PROGRAM P_MotorControl
VAR
	
  	error:BOOL;
    fJogVelocity :LREAL;
	MC_Halt_ServoB: MC_Halt;
	MC_Halt_ServoA: MC_Halt;
	sinGen : FB_singen;	
	ServoA_SPGen: FB_useExtSetpointGen;
	ServoB_SPGen: FB_useExtSetpointGen;
	nSawSPError : INT :=0;
	r_trig_0: r_trig;


	
	b_ExecuteGearIn: BOOL;
	MC_GearInA: MC_GearIn;
	MC_MoveRelativeA: MC_MoveRelative;
	bAbsMoveBExecute: BOOL;
	MC_MoveAbsolute_A: MC_MoveContinuousAbsolute;
	ZeroingReqRtrig: R_TRIG;
	bSetZero: BOOL;
	McWritePArams1: MC_WriteParameterPersistent;
	McWritePArams2: MC_WriteParameterPersistent;
	MC_SetPosition_0: MC_SetPosition;
	MC_SetPosition_1: MC_SetPosition;
	MC_MoveAbsolute_Jog: MC_MoveAbsolute;
	MC_MoveContinuousRelative_0: MC_MoveContinuousRelative;
	MC_MoveRelative_Jog: MC_MoveRelative;
	RelMoveDistance: LREAL;
	bSinGenEnable: BOOL;
	RS_0: rs;
END_VAR
VAR // added by the converter: edge detectors and wires of the graphical bodies
    _rt1 : R_TRIG;
END_VAR

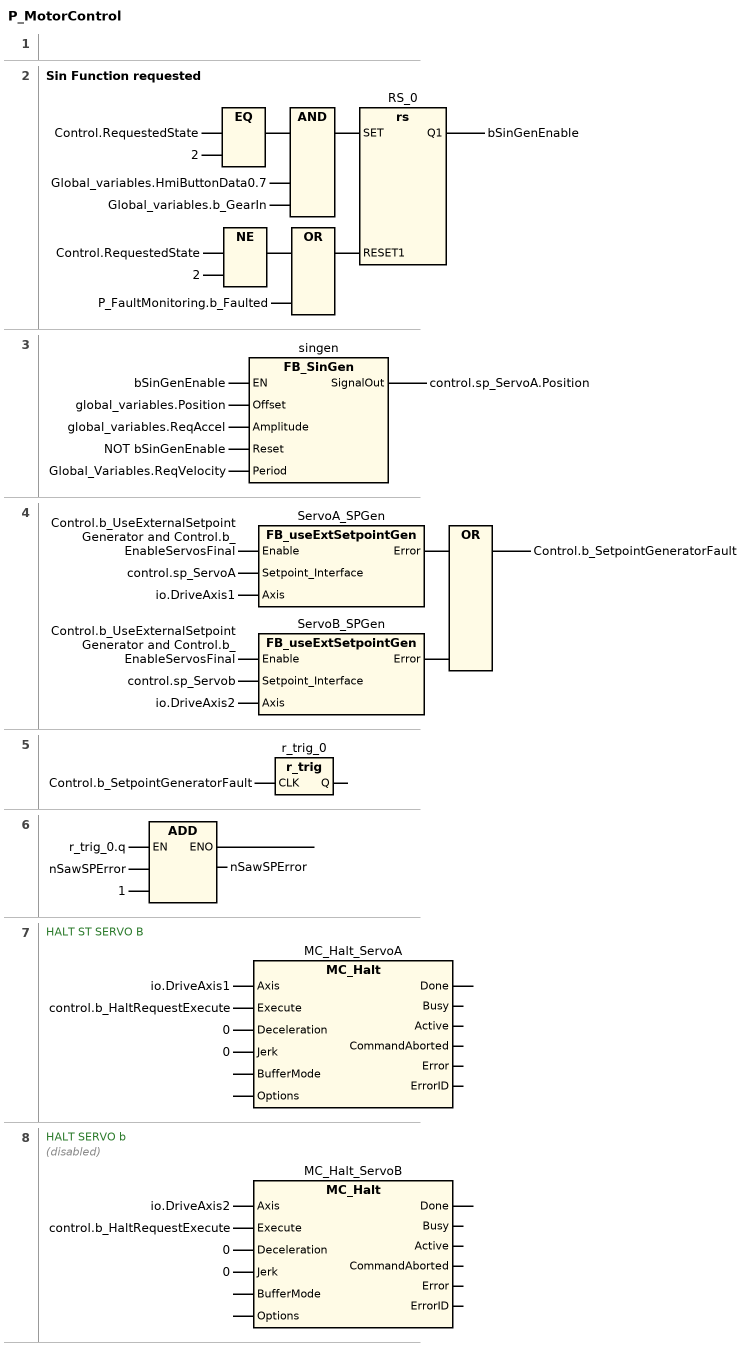
// NETWORK 1

// NETWORK 2: Sin Function requested
RS_0(SET := Control.RequestedState = 2 AND Global_variables.HmiButtonData0.7 AND Global_variables.b_GearIn, RESET1 := Control.RequestedState <> 2 OR P_FaultMonitoring.b_Faulted); // rs
bSinGenEnable := RS_0.Q1;

// NETWORK 3
singen(
    EN := bSinGenEnable,
    Offset := global_variables.Position,
    Amplitude := global_variables.ReqAccel,
    Reset := NOT bSinGenEnable,
    Period := Global_Variables.ReqVelocity); // FB_SinGen
control.sp_ServoA.Position := singen.SignalOut;

// NETWORK 4
ServoA_SPGen(
    Enable := Control.b_UseExternalSetpointGenerator and Control.b_EnableServosFinal,
    Setpoint_Interface := control.sp_ServoA,
    Axis := io.DriveAxis1); // FB_useExtSetpointGen
ServoB_SPGen(
    Enable := Control.b_UseExternalSetpointGenerator and Control.b_EnableServosFinal,
    Setpoint_Interface := control.sp_Servob,
    Axis := io.DriveAxis2); // FB_useExtSetpointGen
Control.b_SetpointGeneratorFault := ServoA_SPGen.Error OR ServoB_SPGen.Error;

// NETWORK 5
r_trig_0(CLK := Control.b_SetpointGeneratorFault); // r_trig

// NETWORK 6
IF r_trig_0.q THEN nSawSPError := nSawSPError + 1; END_IF

// NETWORK 7
// HALT ST SERVO B
MC_Halt_ServoA(Axis := io.DriveAxis1, Execute := control.b_HaltRequestExecute, Deceleration := 0, Jerk := 0); // MC_Halt

// NETWORK 8 (disabled)
// HALT SERVO b
// MC_Halt_ServoB(Axis := io.DriveAxis2, Execute := control.b_HaltRequestExecute, Deceleration := 0, Jerk := 0); // MC_Halt

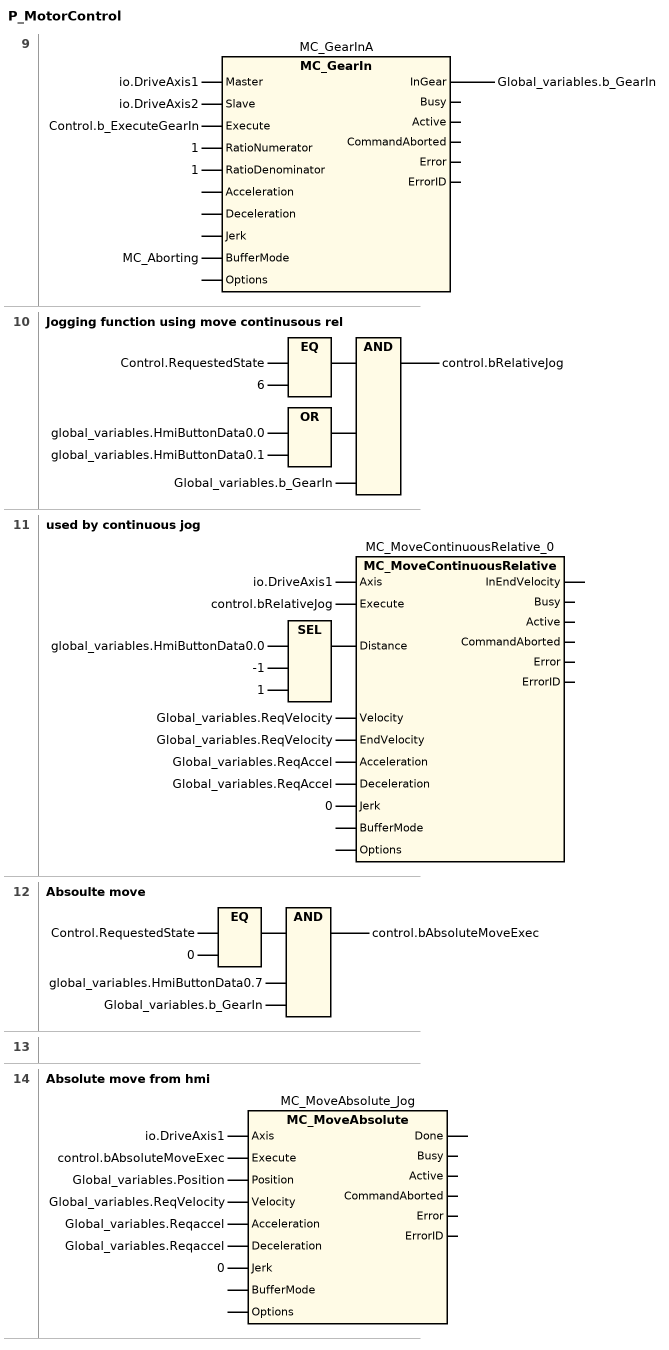
// NETWORK 9
MC_GearInA(
    Master := io.DriveAxis1,
    Slave := io.DriveAxis2,
    Execute := Control.b_ExecuteGearIn,
    RatioNumerator := 1,
    RatioDenominator := 1,
    BufferMode := MC_Aborting); // MC_GearIn
Global_variables.b_GearIn := MC_GearInA.InGear;

// NETWORK 10: Jogging function using move continusous rel
control.bRelativeJog := Control.RequestedState = 6 AND (global_variables.HmiButtonData0.0 OR global_variables.HmiButtonData0.1) AND Global_variables.b_GearIn;

// NETWORK 11: used by continuous jog
MC_MoveContinuousRelative_0(
    Axis := io.DriveAxis1,
    Execute := control.bRelativeJog,
    Distance := SEL(global_variables.HmiButtonData0.0, -1, 1),
    Velocity := Global_variables.ReqVelocity,
    EndVelocity := Global_variables.ReqVelocity,
    Acceleration := Global_variables.ReqAccel,
    Deceleration := Global_variables.ReqAccel,
    Jerk := 0); // MC_MoveContinuousRelative

// NETWORK 12: Absoulte move
control.bAbsoluteMoveExec := Control.RequestedState = 0 AND global_variables.HmiButtonData0.7 AND Global_variables.b_GearIn;

// NETWORK 13

// NETWORK 14: Absolute move from hmi
MC_MoveAbsolute_Jog(
    Axis := io.DriveAxis1,
    Execute := control.bAbsoluteMoveExec,
    Position := Global_variables.Position,
    Velocity := Global_variables.ReqVelocity,
    Acceleration := Global_variables.Reqaccel,
    Deceleration := Global_variables.Reqaccel,
    Jerk := 0); // MC_MoveAbsolute

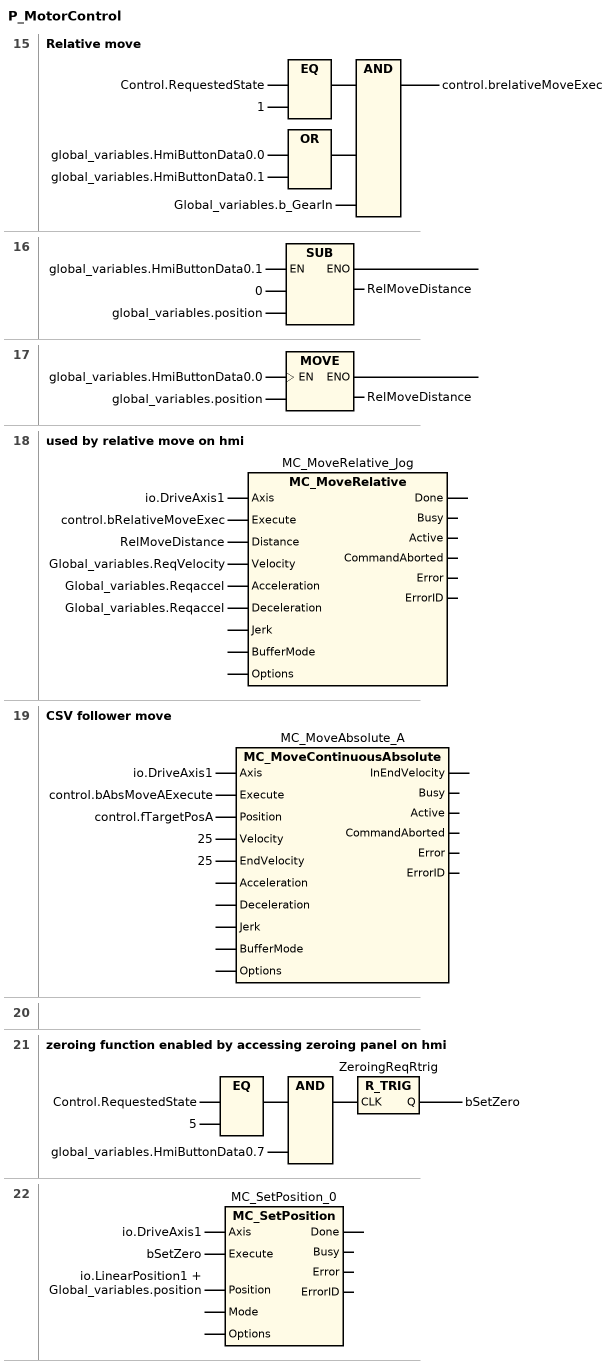
// NETWORK 15: Relative move
control.brelativeMoveExec := Control.RequestedState = 1 AND (global_variables.HmiButtonData0.0 OR global_variables.HmiButtonData0.1) AND Global_variables.b_GearIn;

// NETWORK 16
IF global_variables.HmiButtonData0.1 THEN RelMoveDistance := 0 - global_variables.position; END_IF

// NETWORK 17
_rt1(CLK := global_variables.HmiButtonData0.0);
IF _rt1.Q THEN RelMoveDistance := global_variables.position; END_IF

// NETWORK 18: used by relative move on hmi
MC_MoveRelative_Jog(
    Axis := io.DriveAxis1,
    Execute := control.bRelativeMoveExec,
    Distance := RelMoveDistance,
    Velocity := Global_variables.ReqVelocity,
    Acceleration := Global_variables.Reqaccel,
    Deceleration := Global_variables.Reqaccel); // MC_MoveRelative

// NETWORK 19: CSV follower move
MC_MoveAbsolute_A(
    Axis := io.DriveAxis1,
    Execute := control.bAbsMoveAExecute,
    Position := control.fTargetPosA,
    Velocity := 25,
    EndVelocity := 25); // MC_MoveContinuousAbsolute

// NETWORK 20

// NETWORK 21: zeroing function enabled by accessing zeroing panel on hmi
ZeroingReqRtrig(CLK := Control.RequestedState = 5 AND global_variables.HmiButtonData0.7); // R_TRIG
bSetZero := ZeroingReqRtrig.Q;

// NETWORK 22
MC_SetPosition_0(
    Axis := io.DriveAxis1,
    Execute := bSetZero,
    Position := io.LinearPosition1 + Global_variables.position); // MC_SetPosition

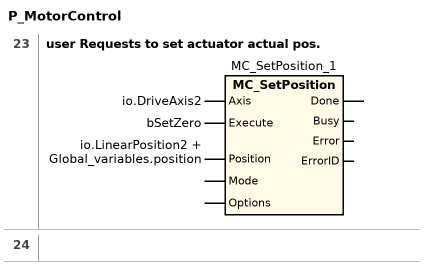
// NETWORK 23: user Requests to set actuator actual pos.
MC_SetPosition_1(
    Axis := io.DriveAxis2,
    Execute := bSetZero,
    Position := io.LinearPosition2 + Global_variables.position); // MC_SetPosition

// NETWORK 24

END_PROGRAM

(* stored: Version 1.1.0.1, ProductVersion 3.1.4024.4
   POU P_MotorControl: Id {a8ffc1f5-463c-4b24-9e55-2df4bd795b0c}, SpecialFunc None *)
